FUNCTION_BLOCK StatusManagement (* Basic Function Block Type *)
  (* Standard: 61499-2 *)
  (* Version 0.0, 2015-05-21, 4DIAC-IDE, 4DIAC-Consortium *)
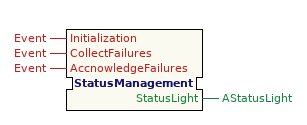
  EVENT_INPUT
    Initialization;
    CollectFailures; (* Initialization Request *)
    AccnowledgeFailures; (* Normal Execution Request *)
  END_EVENT
  PLUGS
    StatusLight : AStatusLight;
  END_PLUGS
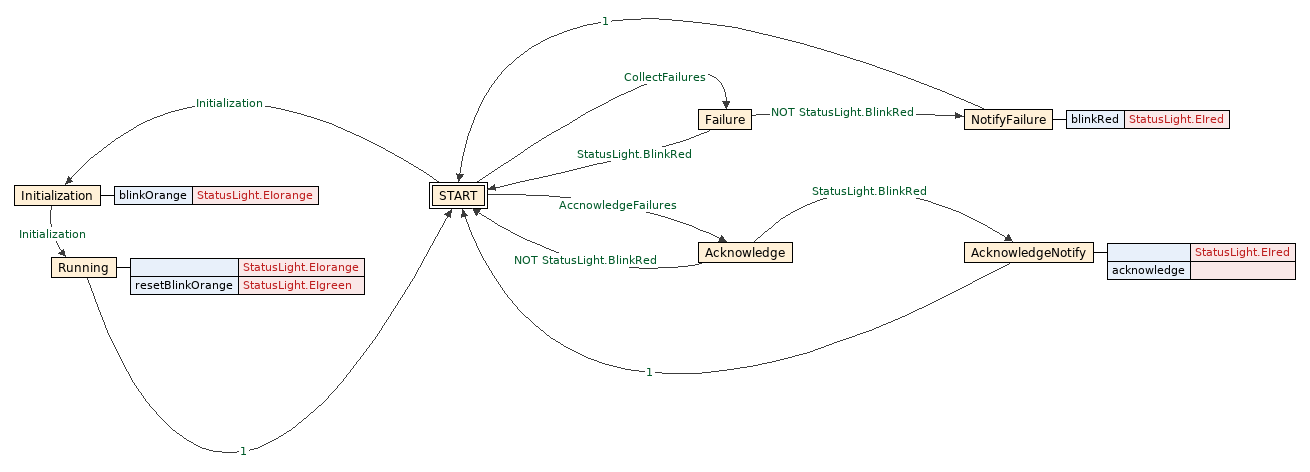
  EC_STATES
    START; (* Initial State *)
    Failure; (* Initialization *)
    AcknowledgeNotify : -> StatusLight.EIred, acknowledge; (* Normal execution *)
    NotifyFailure : blinkRed -> StatusLight.EIred;
    Acknowledge;
    Initialization : blinkOrange -> StatusLight.EIorange;
    Running : -> StatusLight.EIorange, resetBlinkOrange -> StatusLight.EIgreen;
  END_STATES
  EC_TRANSITIONS
    START TO Failure := CollectFailures;
    Failure TO START := StatusLight.BlinkRed;
    AcknowledgeNotify TO START := 1;
    Failure TO NotifyFailure := NOT StatusLight.BlinkRed;
    START TO Acknowledge := AccnowledgeFailures;
    NotifyFailure TO START := 1;
    Acknowledge TO AcknowledgeNotify := StatusLight.BlinkRed;
    Acknowledge TO START := NOT StatusLight.BlinkRed;
    START TO Initialization := Initialization;
    Running TO START := 1;
    Initialization TO Running := Initialization;
  END_TRANSITIONS
  ALGORITHM blinkRed IN ST: (* Normally executed algorithm *)
StatusLight.BlinkRed := true;
  END_ALGORITHM
  ALGORITHM acknowledge IN ST: (* new algorithm *)
StatusLight.BlinkRed := false;
  END_ALGORITHM
  ALGORITHM blinkOrange IN ST: (* new algorithm *)
StatusLight.BlinkOrange := true;
  END_ALGORITHM
  ALGORITHM resetBlinkOrange IN ST: (* new algorithm *)
StatusLight.BlinkRed := false;
  END_ALGORITHM
END_FUNCTION_BLOCK
